FUNCTION_BLOCK FB_JobEventCyclicOutput IMPLEMENTS I_Observer
VAR_OUTPUT
	event_message : ST_JobEventMessage;
END_VAR
VAR
	queue : FB_EventMessageQueue;
	cycle_counter : UINT;
END_VAR

IF queue.usage > 0 THEN
	event_message := queue.get();
END_IF

METHOD notify : BOOL
VAR_INPUT
	publisher	: I_Observable;
END_VAR
VAR_INST
	_event_message : ST_JobEventMessage;
END_VAR
VAR
	job_report : I_JobInfo;
	container : InterfaceContainer;
	num_of_jobs : UDINT;
END_VAR
IF NOT __QUERYINTERFACE(publisher, job_report) THEN
	RETURN;
END_IF

IF job_report.job <> 0 AND_THEN __QUERYINTERFACE(job_report.job.future, container) THEN
	num_of_jobs := container.num_of_jobs;
ELSE
	num_of_jobs := 0;
END_IF

_event_message.job_id := job_report.job.uid;
_event_message.job_namespace := job_report.job.namespace;
_event_message.num_of_job := num_of_jobs;
_event_message.new_state := TO_STRING(job_report.new_state);
_event_message.old_state := TO_STRING(job_report.last_state);
_event_message.record_time := job_report.record_time;
_event_message.subject := job_report.job.future.future_name;
queue.put(_event_message);
notify := TRUE;
END_METHOD

END_FUNCTION_BLOCK

(* stored: Version 1.1.0.1, ProductVersion 3.1.4026.13
   POU FB_JobEventCyclicOutput: Id {9c0d3885-b004-4a83-92db-ed3f004b38ca}, SpecialFunc None
   Method notify: Id {79b5858d-145b-4660-857a-78a4dfda7730} *)
